// TIA Portal V21 export
// export: ExportSetting WithDefaults, DisplayName Totally Integrated Automation Portal, DisplayVersion V21, DisplayName STEP 7 Professional, DisplayVersion V21
FUNCTION "LAD_StartStop" : Void   // FC11, LAD
TITLE = LAD_StartStop
{ S7_Optimized_Access := 'TRUE' }
VERSION : 0.1
// ladder start stop
// stored: AutoNumber true, IsIECCheckEnabled true, SetENOAutomatically false, UDAEnableTagReadback false
   VAR_INPUT
      Start : Bool;
      Stop : Bool;
   END_VAR
   VAR_OUTPUT
      Motor : Bool;
   END_VAR
BEGIN

REGION Network 1: start stop ladder
   // network 1
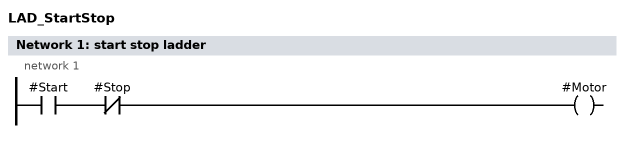
   RUNG wire#powerrail
      Contact( #Start )
      I_Contact( #Stop )
      Coil( #Motor )
   END_RUNG
   // the same network as SCL:
   #Motor := #Start AND NOT #Stop;
END_REGION
END_FUNCTION
